(*
SPDX-FileCopyrightText: © 2026 Oleksandr Tiutyk <trofimich@gmail.com>
SPDX-License-Identifier: MIT
License: https://opensource.org/license/mit
*)

(*!
<summary>Releases every task's auto-dispose registry during application teardown.</summary>
<description>
The runtime must have stopped cyclic execution before FB_exit. This is not a cyclic cleanup entry point.
</description>
*)

FUNCTION_BLOCK INTERNAL MemoryCleanupHelper

(*!
<summary>Clears all task payloads and releases all registered objects and registry buffers.</summary>
<description>
Called by the runtime with cyclic execution stopped. Cleanup callbacks must not throw or register objects. The
return value is not evaluated.
</description>
*)

//!<param name="bInCopyCode">
//! TRUE: the exit method is called in order to leave the instance which will be copied afterwards (online
//! change).
//! </param>

METHOD FB_Exit: BOOL
VAR_INPUT
    bInCopyCode: BOOL;  
END_VAR
DynamicMemoryManager.CleanupAllTasks();
END_METHOD

END_FUNCTION_BLOCK

(* stored: Version 1.1.0.1
   POU MemoryCleanupHelper: Id {7dc830f2-0958-4a4b-8a4a-b4858028b05f}, SpecialFunc None
   Method FB_Exit: Id {ab8a9fe6-b7e4-4631-afbd-30ad2c87a604} *)
